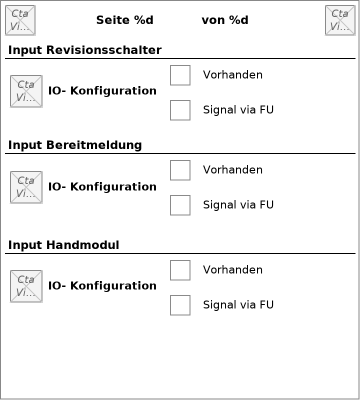
VISUALIZATION VIS_VERDICHTER_PARAMETER_IO  // 360x400
VAR_INPUT
    ITF_VERDICHTERIN : ITF_VERDICHTER;
END_VAR
VAR
    uiPage  :   UINT;
    uiMin   :   UINT    := 0;
    uiMax   :   UINT    := 4
;
END_VAR
    Frame (0,40 360x360), frame switch variable: uiPage
        shows VIS_VERDICHTER_PARAMETER_IO0(ITF_VERDICHTERIN := ITF_VERDICHTERIN, ITF_RevSwitch_IN := ITF_VERDICHTERIN.proRevisionSwitch_ITF, ITF_VerdiReady_IN := ITF_VERDICHTERIN.proReady_ITF, ITF_VerdiHandMod_IN := ITF_VERDICHTERIN.proHandModul_ITF)
        shows VIS_VERDICHTER_PARAMETER_IO1(ITF_VERDICHTERIN := ITF_VERDICHTERIN, ITF_VerdichterOn_IN := ITF_VERDICHTERIN.proIsOn_ITF)
        shows VIS_VERDICHTER_PARAMETER_IO2(ITF_VERDICHTERIN := ITF_VERDICHTERIN, ITF_VerdiNoError_IN := ITF_VERDICHTERIN.proNoError_ITF)
        shows VIS_VERDICHTER_PARAMETER_IO3(ITF_VERDICHTERIN := ITF_VERDICHTERIN, ITF_ActualValue_IN := ITF_VERDICHTERIN.proActualValue_ITF)
        shows VIS_VERDICHTER_PARAMETER_IO4(ITF_VERDICHTERIN := ITF_VERDICHTERIN, ITF_xOn_IN := ITF_VERDICHTERIN.proOn_ITF, ITF_rOnY_IN := ITF_VERDICHTERIN.proOnY_ITF)
    Image (325,5 30x30), invisible if: uiPage = uiMax, image: CtaVisSymbols.ImagePool.arrow-right_square
        OnMouseClick: execute {
            uiPage := uiPage + 1;
            IF uiPage >= uiMax THEN
                uiPage := uiMax;
            END_IF;
        }
    Image (5,5 30x30), invisible if: uiPage = uiMin, image: CtaVisSymbols.ImagePool.arrow-left_square
        OnMouseClick: execute {
            uiPage := uiPage - 1;
            IF uiPage <= uiMin THEN
                uiPage := uiMin;
            END_IF;
        }
    Textfield (175,5 100x30), "von %d", text variable: uiMax
    Textfield (75,5 100x30), "Seite %d", text variable: uiPage
END_VISUALIZATION

// 40 Visualizations/POPUP/PARAMETER/VERDICHTER_IO/VIS_VERDICHTER_PARAMETER_IO2
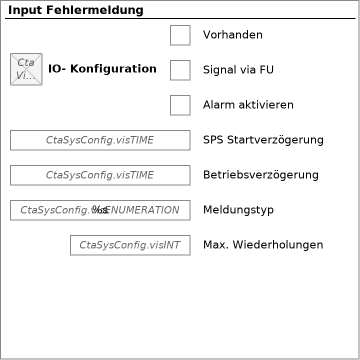
VISUALIZATION VIS_VERDICHTER_PARAMETER_IO2  // 360x360
VAR_INPUT
    ITF_VERDICHTERIN 		:	ITF_VERDICHTER;
	ITF_VerdiNoError_IN		:	CtaSysIO.ITF_IO;
END_VAR
    Label (5,0 350x20), "Input Fehlermeldung"
    Frame (170,25 20x20)
        shows CtaSysConfig.visBOOL(visfbBOOLIn := ITF_VERDICHTERIN.P_scIO_IsNoError_fbxEnable)
    Label (200,25 150x20), "Vorhanden"
    Frame (170,60 20x20)
        shows CtaSysConfig.visBOOL(visfbBOOLIn := ITF_VERDICHTERIN.P_scIO_IsNoError_fbxInputMb)
    Label (200,60 150x20), "Signal via FU"
    Frame (170,95 20x20)
        shows CtaSysConfig.visBOOL(visfbBOOLIn := ITF_VERDICHTERIN.P_scIO_IsNoError_fbxDoesAlarm)
    Label (200,95 150x20), "Alarm aktivieren"
    Frame (10,130 180x20)
        shows CtaSysConfig.visTIME(visfbTIMEIn := ITF_VERDICHTERIN.P_scIO_IsNoError_fbtDelayStartSps)
    Label (200,130 150x20), "SPS Startverzögerung"
    Label (200,165 150x20), "Betriebsverzögerung"
    Frame (10,165 180x20)
        shows CtaSysConfig.visTIME(visfbTIMEIn := ITF_VERDICHTERIN.P_scIO_IsNoError_fbtDelayRun)
    Label (200,200 150x20), "Meldungstyp"
    Label (200,235 150x20), "Max. Wiederholungen"
    Line (5,18) (355,18)
    Frame (70,235 120x20)
        shows CtaSysConfig.visINT(visfbINTIn := ITF_VERDICHTERIN.P_scIO_IsNoError_fbiMaxErrorRetryAllowed)
    Frame (10,200 180x20)
        shows CtaSysConfig.visENUMERATION(visfbENUIn := ITF_VERDICHTERIN.P_scIO_IsNoError_fbiTypeOfAck)
    Image (10,53 32x32), invisible if: ITF_VerdiNoError_IN = 0, image: CtaVisSymbols.ImagePool.build
        OnMouseDown:  Dialog=VIS_ANTRIEB_POPUP_IO_ITF, Parameters={ITF_IO_IN: ITF_VerdiNoError_IN}, OpenModal=True, OpenCentered=True
    Label (45,59 120x20), "IO- Konfiguration", invisible if: ITF_VerdiNoError_IN = 0
    Textfield (30,200 140x20), "%s", text list: 'CtaAppReport.txtLibAp99_2enTypeOfAck', text index: CtaSysConfig.fcGetEnumerationId(ITF_VERDICHTERIN.P_scIO_IsNoError_fbiTypeOfAck)
END_VISUALIZATION

// 40 Visualizations/POPUP/PARAMETER/VERDICHTER_IO/VIS_VERDICHTER_PARAMETER_IO3
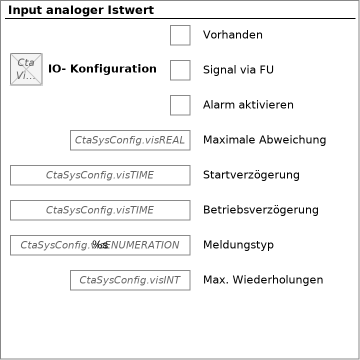
VISUALIZATION VIS_VERDICHTER_PARAMETER_IO3  // 360x360
VAR_INPUT
    ITF_VERDICHTERIN 	:	ITF_VERDICHTER;
	ITF_ActualValue_IN	:	CtaSysIO.ITF_IO;
END_VAR
    Label (5,0 350x20), "Input analoger Istwert"
    Frame (170,25 20x20)
        shows CtaSysConfig.visBOOL(visfbBOOLIn := ITF_VERDICHTERIN.P_scIO_IsValue_fbxEnable)
    Label (200,25 150x20), "Vorhanden"
    Frame (170,60 20x20)
        shows CtaSysConfig.visBOOL(visfbBOOLIn := ITF_VERDICHTERIN.P_scIO_IsValue_fbxInputMb)
    Label (200,60 150x20), "Signal via FU"
    Frame (170,95 20x20)
        shows CtaSysConfig.visBOOL(visfbBOOLIn := ITF_VERDICHTERIN.P_scIO_IsValue_fbxDoesAlarm)
    Label (200,95 150x20), "Alarm aktivieren"
    Frame (10,165 180x20)
        shows CtaSysConfig.visTIME(visfbTIMEIn := ITF_VERDICHTERIN.P_scIO_IsValue_fbtDelayStart)
    Label (200,165 150x20), "Startverzögerung"
    Label (200,200 150x20), "Betriebsverzögerung"
    Frame (10,200 180x20)
        shows CtaSysConfig.visTIME(visfbTIMEIn := ITF_VERDICHTERIN.P_scIO_IsValue_fbtDelayRun)
    Frame (70,130 120x20)
        shows CtaSysConfig.visREAL(visfbREALIn := ITF_VERDICHTERIN.P_scIO_IsValue_fbrMaxDiff)
    Label (200,130 150x20), "Maximale Abweichung"
    Label (200,235 150x20), "Meldungstyp"
    Label (200,270 150x20), "Max. Wiederholungen"
    Line (5,18) (355,18)
    Frame (70,270 120x20)
        shows CtaSysConfig.visINT(visfbINTIn := ITF_VERDICHTERIN.P_scIO_IsValue_fbiMaxErrorRetryAllowed)
    Frame (10,235 180x20)
        shows CtaSysConfig.visENUMERATION(visfbENUIn := ITF_VERDICHTERIN.P_scIO_IsValue_fbiTypeOfAck)
    Image (10,53 32x32), invisible if: ITF_ActualValue_IN = 0, image: CtaVisSymbols.ImagePool.build
        OnMouseDown:  Dialog=VIS_ANTRIEB_POPUP_IO_ITF, Parameters={ITF_IO_IN: ITF_ActualValue_IN}, OpenModal=True, OpenCentered=True
    Label (45,59 120x20), "IO- Konfiguration", invisible if: ITF_ActualValue_IN = 0
    Textfield (30,235 140x20), "%s", text list: 'CtaAppReport.txtLibAp99_2enTypeOfAck', text index: CtaSysConfig.fcGetEnumerationId(ITF_VERDICHTERIN.P_scIO_IsValue_fbiTypeOfAck)
END_VISUALIZATION

// 40 Visualizations/POPUP/PARAMETER/VERDICHTER_InfluxDb/VIS_VERDICHTER_PARAMETER_TRENDLOG
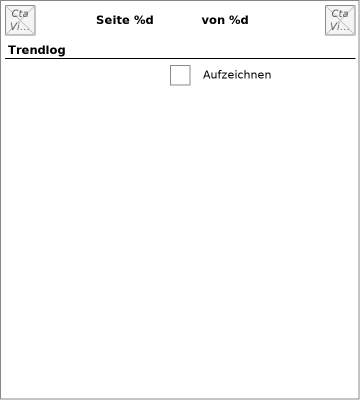
VISUALIZATION VIS_VERDICHTER_PARAMETER_TRENDLOG  // 360x400
VAR_INPUT
    ITF_VERDICHTERIN : ITF_VERDICHTER;
END_VAR
VAR
    uiPage  :   UINT;
    uiMin   :   UINT    := 0;
    uiMax   :   UINT    := 0;
END_VAR
    Image (5,5 30x30), invisible if: uiPage = uiMin, image: CtaVisSymbols.ImagePool.arrow-left_square
        OnMouseClick: execute {
            uiPage := uiPage - 1;
            IF uiPage <= uiMin THEN
                uiPage := uiMin;
            END_IF;
        }
    Image (325,5 30x30), invisible if: uiPage = uiMax, image: CtaVisSymbols.ImagePool.arrow-right_square
        OnMouseClick: execute {
            uiPage := uiPage + 1;
            IF uiPage >= uiMax THEN
                uiPage := uiMax;
            END_IF;
        }
    Frame (0,40 360x360), frame switch variable: uiPage
        shows VIS_VERDICHTER_PARAMETER_TRENDLOG0(ITF_VERDICHTERIN := ITF_VERDICHTERIN)
        shows AT_ParameterIO1(ITF_Parameter := ITF_Parameter)
        pReferences[0]: ITF_Parameter=ITF_Parameter
    Textfield (75,5 100x30), "Seite %d", text variable: uiPage
    Textfield (175,5 100x30), "von %d", text variable: uiMax
END_VISUALIZATION

// 40 Visualizations/POPUP/PARAMETER/VERDICHTER_InfluxDb/VIS_VERDICHTER_PARAMETER_TRENDLOG0
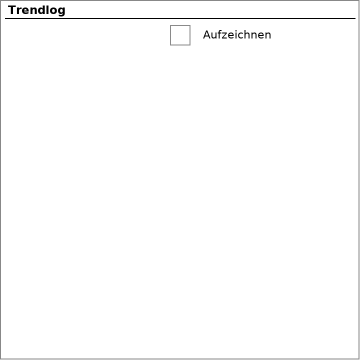
VISUALIZATION VIS_VERDICHTER_PARAMETER_TRENDLOG0  // 360x360
VAR_INPUT
    ITF_VERDICHTERIN : ITF_VERDICHTER;
END_VAR
    Frame (170,25 20x20)
        shows CtaSysConfig.visBOOL(visfbBOOLIn := ITF_VERDICHTERIN.P_scInfluxDb_fbxEnable)
    Label (200,25 150x20), "Aufzeichnen"
    Label (5,0 350x20), "Trendlog"
    Line (5,18) (355,18)
END_VISUALIZATION

// 40 Visualizations/POPUP/IO/VIS_VERDICHTER_IO0
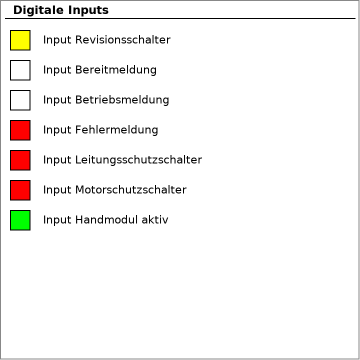
VISUALIZATION VIS_VERDICHTER_IO0  // 360x360
VAR_INPUT
    ITF_VERDICHTERIN    :   ITF_VERDICHTER;	
END_VAR
    Label (40,30 320x20), "Input Revisionsschalter", invisible if: ITF_VERDICHTERIN.proNotShowDI_RevisionSwitchOk
    Label (40,60 320x20), "Input Bereitmeldung", invisible if: ITF_VERDICHTERIN.proNotShowDI_Ready
    Rectangle (10,30 20x20), colour toggle: ITF_VERDICHTERIN.proGetDI_RevisionSwitchOK, invisible if: ITF_VERDICHTERIN.proNotShowDI_RevisionSwitchOk
    Rectangle (10,60 20x20), colour toggle: ITF_VERDICHTERIN.proGetDI_IsReady, invisible if: ITF_VERDICHTERIN.proNotShowDI_Ready
    Label (40,120 320x20), "Input Fehlermeldung", invisible if: ITF_VERDICHTERIN.proNotShowDI_NoError
    Rectangle (10,120 20x20), colour toggle: ITF_VERDICHTERIN.proGetDI_NoError, invisible if: ITF_VERDICHTERIN.proNotShowDI_NoError
    Rectangle (10,150 20x20), colour toggle: ITF_VERDICHTERIN.proGetDI_FuseOK, invisible if: ITF_VERDICHTERIN.proNotShowDI_FuseOk
    Label (40,150 320x20), "Input Leitungsschutzschalter", invisible if: ITF_VERDICHTERIN.proNotShowDI_FuseOk
    Label (40,180 320x20), "Input Motorschutzschalter", invisible if: ITF_VERDICHTERIN.proNotShowDI_VerdichterFuseOk
    Rectangle (10,180 20x20), colour toggle: ITF_VERDICHTERIN.proGetDI_VerdichterFuseOk, invisible if: ITF_VERDICHTERIN.proNotShowDI_VerdichterFuseOk
    Label (40,210 320x20), "Input Handmodul aktiv", invisible if: ITF_VERDICHTERIN.proNotShowDI_VerdichterHand
    Rectangle (10,210 20x20), colour toggle: ITF_VERDICHTERIN.proGetDI_VerdichterHand, invisible if: ITF_VERDICHTERIN.proNotShowDI_VerdichterHand
    Label (40,90 320x20), "Input Betriebsmeldung", invisible if: ITF_VERDICHTERIN.proNotShowDI_IsOn
    Rectangle (10,90 20x20), colour toggle: ITF_VERDICHTERIN.proGetDI_IsOn, invisible if: ITF_VERDICHTERIN.proNotShowDI_IsOn
    Label (10,0 350x20), "Digitale Inputs"
    Line (5,18) (355,18)
END_VISUALIZATION

// 40 Visualizations/POPUP/IO/VIS_VERDICHTER_IO
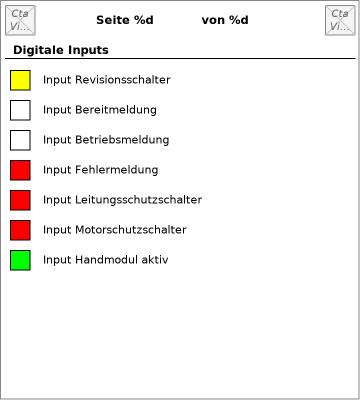
VISUALIZATION VIS_VERDICHTER_IO  // 360x400
VAR_INPUT
    ITF_VERDICHTERIN    :   ITF_VERDICHTER;	
END_VAR
VAR
    uiPage  :   UINT;
    uiMin   :   UINT    := 0;
    uiMax   :   UINT    := 1;
END_VAR
    Frame (0,40 360x360), frame switch variable: uiPage
        shows VIS_VERDICHTER_IO0(ITF_VERDICHTERIN := ITF_VERDICHTERIN)
        shows VIS_VERDICHTER_IO1(ITF_VERDICHTERIN := ITF_VERDICHTERIN)
        shows AT_ParameterIO2(ITF_Parameter := ITF_Parameter)
        shows AT_ParameterIO3(ITF_Parameter := ITF_Parameter)
    Image (325,5 30x30), invisible if: uiPage = uiMax, image: CtaVisSymbols.ImagePool.arrow-right_square
        OnMouseClick: execute {
            uiPage := uiPage + 1;
            IF uiPage >= uiMax THEN
                uiPage := uiMax;
            END_IF;
        }
    Image (5,5 30x30), invisible if: uiPage = uiMin, image: CtaVisSymbols.ImagePool.arrow-left_square
        OnMouseClick: execute {
            uiPage := uiPage - 1;
            IF uiPage <= uiMin THEN
                uiPage := uiMin;
            END_IF;
        }
    Textfield (175,5 100x30), "von %d", text variable: uiMax
    Textfield (75,5 100x30), "Seite %d", text variable: uiPage
END_VISUALIZATION

// 40 Visualizations/POPUP/IO/VIS_VERDICHTER_IO1
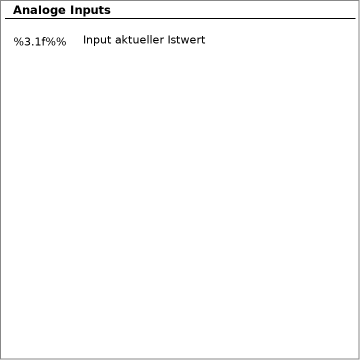
VISUALIZATION VIS_VERDICHTER_IO1  // 360x360
VAR_INPUT
    ITF_VERDICHTERIN    :   ITF_VERDICHTER;	
END_VAR
    Label (80,30 280x20), "Input aktueller Istwert", invisible if: ITF_VERDICHTERIN.proNotShowAI_ActualValue
    Label (10,0 350x20), "Analoge Inputs"
    Textfield (10,32 60x20), "%3.1f%%", text variable: ITF_VERDICHTERIN.proGetAI_ActualValue, invisible if: ITF_VERDICHTERIN.proNotShowAI_ActualValue
    Line (5,18) (355,18)
END_VISUALIZATION

// 40 Visualizations/ICON/VERDICHTER_BASE/VALUE/ValueUpDwn
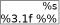
VISUALIZATION ValueUpDwn  // 60x25
VAR_INPUT
    ITF_VERDICHTER_IN   :   ITF_VERDICHTER;	
END_VAR
VAR_INPUT CONSTANT
    uiTextAusrichtung   : UINT := 4;    // 0 = Oben links | 1 = Horizontal zentriert | 2 = Rechts | 4 = Vertikal zentriert | 8 = Unten
END_VAR
    Textfield (0,0 60x12), "%s", text variable: ITF_VERDICHTER_IN.proGetBMK, invisible if: ITF_VERDICHTER_IN.proNoBmkInList
        p3718999670: uiTextAusrichtung
    Textfield (0,13 60x12), "%3.1f %%", text variable: ITF_VERDICHTER_IN.proLeistung, invisible if: NOT ITF_VERDICHTER_IN.proIsRegulatet
        p3718999670: uiTextAusrichtung
END_VISUALIZATION

// 40 Visualizations/ICON/VERDICHTER_LEFT/VERDICHTER_LEFT_ABOVE/VIS_VERDICHTER_LEFT_ABOVE
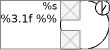
VISUALIZATION VIS_VERDICHTER_LEFT_ABOVE  // 110x50
VAR_INPUT
    ITF_VERDICHTER_IN   :   ITF_VERDICHTER;	
END_VAR
VAR_INPUT CONSTANT
    stExklParameter		:   STRING[40] := '';	
END_VAR
VAR CONSTANT
	uiIconnr		:	UINT := 0;
END_VAR
    Frame (0,0 110x50), invisible if: NOT fcCheckQuerryAndIconReturn(_ITF_IN := ITF_VERDICHTER_IN, _uiIconNr_IN := uiIconNr)
        shows VIS_VERDICHTER_LeftAboveCheckQuerry(ITF_VERDICHTER_IN := ITF_VERDICHTER_IN, stExklParameter := stExklParameter)
END_VISUALIZATION

// 40 Visualizations/ICON/VERDICHTER_LEFT/VERDICHTER_LEFT_ABOVE/VIS_VERDICHTER_LeftAboveCheckIsEnabled
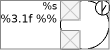
VISUALIZATION VIS_VERDICHTER_LeftAboveCheckIsEnabled  // 110x50
VAR_INPUT
    ITF_VERDICHTER_IN   :   ITF_VERDICHTER;	
    stExklParameter		:   STRING[40];	
END_VAR
    Frame (60,0 50x50), invisible if: NOT ITF_VERDICHTER_IN.proIsEnabled
        shows Icon_Left(ITF_VERDICHTER_IN := ITF_VERDICHTER_IN)
    Frame (0,0 60x25), invisible if: NOT ITF_VERDICHTER_IN.proIsEnabled
        shows ValueUpDwn(ITF_VERDICHTER_IN := ITF_VERDICHTER_IN, uiTextAusrichtung := 6)
    Frame (95,0 15x15), invisible if: NOT ITF_VERDICHTER_IN.proIsEnabled
        shows CommandOn(ITF_VERDICHTER_IN := ITF_VERDICHTER_IN)
    Rectangle (0,0 110x50)
        OnMouseClick:  Dialog=POPUP_VERDICHTER, Parameters={stExklParameter: stExklParameter, ITF_VERDICHTERIN: ITF_VERDICHTER_IN, uiPopUpGruppe: 0}, OpenCentered=True
END_VISUALIZATION

// 40 Visualizations/ICON/VERDICHTER_LEFT/VERDICHTER_LEFT_ABOVE/VIS_VERDICHTER_LeftAboveCheckQuerry
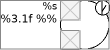
VISUALIZATION VIS_VERDICHTER_LeftAboveCheckQuerry  // 110x50
VAR_INPUT
    ITF_VERDICHTER_IN   :   ITF_VERDICHTER;	
    stExklParameter		:   STRING[40];	
END_VAR
    Frame (0,0 110x50)
        shows VIS_VERDICHTER_LeftAboveCheckIsEnabled(ITF_VERDICHTER_IN := ITF_VERDICHTER_IN, stExklParameter := stExklParameter)
END_VISUALIZATION

// 40 Visualizations/ICON/VERDICHTER_LEFT/VERDICHTER_LEFT_BELOW/VIS_VERDICHTER_LEFT_BELOW
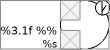
VISUALIZATION VIS_VERDICHTER_LEFT_BELOW  // 110x50
VAR_INPUT
    ITF_VERDICHTER_IN   :   ITF_VERDICHTER;	
END_VAR
VAR_INPUT CONSTANT
    stExklParameter		:   STRING[40] := '';	
END_VAR
VAR CONSTANT
	uiIconNr		:	UINT := 1 ;
END_VAR
    Frame (0,0 110x50), invisible if: NOT fcCheckQuerryAndIconReturn(_ITF_IN := ITF_VERDICHTER_IN, _uiIconNr_IN := uiIconNr)
        shows VIS_VERDICHTER_LeftBelowCheckQuerry(ITF_VERDICHTER_IN := ITF_VERDICHTER_IN, stExklParameter := stExklParameter)
END_VISUALIZATION

// 40 Visualizations/ICON/VERDICHTER_LEFT/VERDICHTER_LEFT_BELOW/VIS_VERDICHTER_LeftBelowCheckIsEnabled
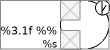
VISUALIZATION VIS_VERDICHTER_LeftBelowCheckIsEnabled  // 110x50
VAR_INPUT
    ITF_VERDICHTER_IN   :   ITF_VERDICHTER;	
    stExklParameter		:   STRING[40];	
END_VAR
    Frame (60,0 50x50), invisible if: NOT ITF_VERDICHTER_IN.proIsEnabled
        shows Icon_Left(ITF_VERDICHTER_IN := ITF_VERDICHTER_IN)
    Frame (0,25 60x27), invisible if: NOT ITF_VERDICHTER_IN.proIsEnabled
        shows ValueDwnUp(ITF_VERDICHTER_IN := ITF_VERDICHTER_IN, uiTextAusrichtung := 6)
    Frame (95,0 15x15), invisible if: NOT ITF_VERDICHTER_IN.proIsEnabled
        shows CommandOn(ITF_VERDICHTER_IN := ITF_VERDICHTER_IN)
    Rectangle (0,0 110x50)
        OnMouseClick:  Dialog=POPUP_VERDICHTER, Parameters={stExklParameter: stExklParameter, ITF_VERDICHTERIN: ITF_VERDICHTER_IN, uiPopUpGruppe: 0}, OpenCentered=True
END_VISUALIZATION

// 40 Visualizations/ICON/VERDICHTER_LEFT/VERDICHTER_LEFT_BELOW/VIS_VERDICHTER_LeftBelowCheckQuerry
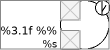
VISUALIZATION VIS_VERDICHTER_LeftBelowCheckQuerry  // 110x50
VAR_INPUT
    ITF_VERDICHTER_IN   :   ITF_VERDICHTER;
    stExklParameter		:   STRING[40];	
END_VAR
    Frame (0,0 110x50)
        shows VIS_VERDICHTER_LeftBelowCheckIsEnabled(ITF_VERDICHTER_IN := ITF_VERDICHTER_IN, stExklParameter := stExklParameter)
END_VISUALIZATION

// 40 Visualizations/ICON/VERDICHTER_RIGHT/VERDICHTER_RIGHT_BELOW/VIS_VERDICHTER_RIGHT_BELOW
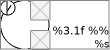
VISUALIZATION VIS_VERDICHTER_RIGHT_BELOW  // 110x50
VAR_INPUT
    ITF_VERDICHTER_IN   :   ITF_VERDICHTER;	
END_VAR
VAR_INPUT CONSTANT
    stExklParameter		:   STRING[40] := '';	
END_VAR
VAR CONSTANT
	uiIconNr		:	UINT := 3;
END_VAR
    Frame (0,0 110x50), invisible if: NOT fcCheckQuerryAndIconReturn(_ITF_IN := ITF_VERDICHTER_IN, _uiIconNr_IN := uiIconNr)
        shows VIS_VERDICHTER_RigthBelowCheckQuerry(ITF_VERDICHTER_IN := ITF_VERDICHTER_IN, stExklParameter := stExklParameter)
END_VISUALIZATION

// 40 Visualizations/ICON/VERDICHTER_RIGHT/VERDICHTER_RIGHT_BELOW/VIS_VERDICHTER_RigthBelowCheckIsEnabled
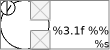
VISUALIZATION VIS_VERDICHTER_RigthBelowCheckIsEnabled  // 110x50
VAR_INPUT
    ITF_VERDICHTER_IN   :   ITF_VERDICHTER;	
    stExklParameter		:   STRING[40];	
END_VAR
    Frame (0,0 50x50), invisible if: NOT ITF_VERDICHTER_IN.proIsEnabled
        shows Icon_Right(ITF_VERDICHTER_IN := ITF_VERDICHTER_IN)
    Frame (52,25 60x27), invisible if: NOT ITF_VERDICHTER_IN.proIsEnabled
        shows ValueDwnUp(ITF_VERDICHTER_IN := ITF_VERDICHTER_IN, uiTextAusrichtung := 4)
    Frame (0,0 15x15), invisible if: NOT ITF_VERDICHTER_IN.proIsEnabled
        shows CommandOn(ITF_VERDICHTER_IN := ITF_VERDICHTER_IN)
    Rectangle (0,0 110x50)
        OnMouseClick:  Dialog=POPUP_VERDICHTER, Parameters={stExklParameter: stExklParameter, ITF_VERDICHTERIN: ITF_VERDICHTER_IN, uiPopUpGruppe: 0}, OpenCentered=True
END_VISUALIZATION

// 40 Visualizations/ICON/VERDICHTER_RIGHT/VERDICHTER_RIGHT_BELOW/VIS_VERDICHTER_RigthBelowCheckQuerry
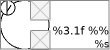
VISUALIZATION VIS_VERDICHTER_RigthBelowCheckQuerry  // 110x50
VAR_INPUT
    ITF_VERDICHTER_IN   :   ITF_VERDICHTER;	
    stExklParameter		:   STRING[40];	
END_VAR
    Frame (0,0 110x50)
        shows VIS_VERDICHTER_RigthBelowCheckIsEnabled(ITF_VERDICHTER_IN := ITF_VERDICHTER_IN, stExklParameter := stExklParameter)
END_VISUALIZATION

// 40 Visualizations/ICON/VERDICHTER_BASE/ICON/Icon_Right
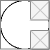
VISUALIZATION Icon_Right  // 50x50
VAR_INPUT
    ITF_VERDICHTER_IN   :   ITF_VERDICHTER;	
END_VAR
    Ellipse (0,0 49x49), colour toggle: ITF_VERDICHTER_IN.proMotorIsOn, invisible if: ITF_VERDICHTER_IN.proIsError
    Ellipse (0,0 49x49), colour toggle: ITF_VERDICHTER_IN.proIsError
    Image (30,0 20x20), invisible if: NOT ITF_VERDICHTER_IN.proIsWarning, image: CtaVisSymbols.ImagePool.CtaWarning
    Image (30,30 20x20), invisible if: NOT ITF_VERDICHTER_IN.proIsHandOnOrOff, image: CtaVisSymbols.ImagePool.front_hand_Yellow
    Image (30,30 20x20), invisible if: NOT ITF_VERDICHTER_IN.proHandOff, image: CtaVisSymbols.ImagePool.front_hand_Yellow_Off
END_VISUALIZATION

// 40 Visualizations/POPUP/PARAMETER/VIS_ANTRIEB_POPUP_IO_ITF
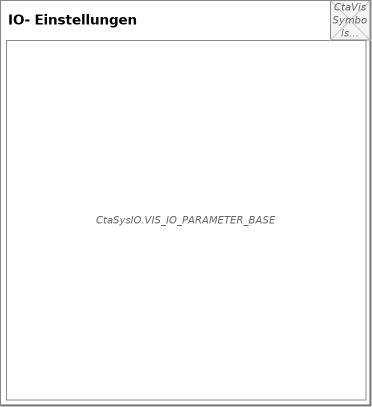
VISUALIZATION VIS_ANTRIEB_POPUP_IO_ITF  // 372x407
VAR_INPUT
    ITF_IO_IN    :   CtaSysIO.ITF_IO;	
END_VAR
    RoundedRectangle (0,0 370x405)
    Frame (6,40 360x360)
        shows CtaSysIO.VIS_IO_PARAMETER_BASE(ITF_IO_IN := ITF_IO_IN)
        shows VIS_ANTRIEB_PARAMETER_IO1(ITF_ANTRIEBIN := ITF_ANTRIEBIN)
        shows VIS_ANTRIEB_PARAMETER_IO2(ITF_ANTRIEBIN := ITF_ANTRIEBIN)
        shows VIS_ANTRIEB_PARAMETER_IO3(ITF_ANTRIEBIN := ITF_ANTRIEBIN)
    Image (330,0 40x40), image: CtaVisSymbols.ImagePool.close_solo_black
        OnMouseClick:  Dialog=VIS_ANTRIEB_POPUP_IO_ITF, Result=None, NumpadKeypadSet=True
    Label (5,0 150x40), "IO- Einstellungen"
END_VISUALIZATION

// 40 Visualizations/POPUP/PARAMETER/VERDICHTER_IO/VIS_VERDICHTER_PARAMETER_IO4
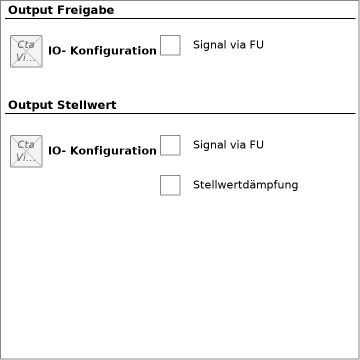
VISUALIZATION VIS_VERDICHTER_PARAMETER_IO4  // 360x360
VAR_INPUT
    ITF_VERDICHTERIN   	:   ITF_VERDICHTER;	
	ITF_xOn_IN			:	CtaSysIO.ITF_IO;
	ITF_rOnY_IN			:	CtaSysIO.ITF_IO;
END_VAR
    Label (5,0 350x20), "Output Freigabe"
    Label (5,95 350x20), "Output Stellwert"
    Line (5,113) (355,113)
    Line (5,18) (355,18)
    Image (10,35 32x32), invisible if: ITF_xOn_IN = 0, image: CtaVisSymbols.ImagePool.build
        OnMouseDown:  Dialog=VIS_ANTRIEB_POPUP_IO_ITF, Parameters={ITF_IO_IN: ITF_xOn_IN}, OpenModal=True, OpenCentered=True
    Image (10,135 32x32), invisible if: ITF_rOnY_IN = 0, image: CtaVisSymbols.ImagePool.build
        OnMouseDown:  Dialog=VIS_ANTRIEB_POPUP_IO_ITF, Parameters={ITF_IO_IN: ITF_rOnY_IN}, OpenModal=True, OpenCentered=True
    Label (45,41 120x20), "IO- Konfiguration", invisible if: ITF_xOn_IN = 0
    Label (45,141 120x20), "IO- Konfiguration", invisible if: ITF_rOnY_IN = 0
    Frame (160,35 20x20)
        shows CtaSysConfig.visBOOL(visfbBOOLIn := ITF_VERDICHTERIN.P_scFU_fbxReleaseMb)
    Label (190,35 150x20), "Signal via FU"
    Frame (160,135 20x20)
        shows CtaSysConfig.visBOOL(visfbBOOLIn := ITF_VERDICHTERIN.P_scFU_fbxSollWertMb)
    Label (190,135 150x20), "Signal via FU"
    Label (190,175 150x20), "Stellwertdämpfung"
    Frame (160,175 20x20)
        shows CtaAppDumper.VisDumperSmall(fbDumper := ITF_VERDICHTERIN.proRefToRonYDumper)
END_VISUALIZATION

// 40 Visualizations/POPUP/OVERVIEW/ResetVerdiTime
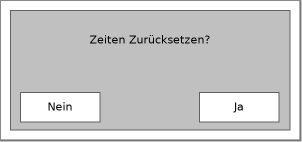
VISUALIZATION ResetVerdiTime  // 302x142
VAR_IN_OUT
	ITF_VERDICHTER_IN		:		ITF_VERDICHTER;
END_VAR
    RoundedRectangle (0,0 300x140)
    RoundedRectangle (10,10 280x120)
    Label (50,10 200x60), "Zeiten Zurücksetzen?"
    RoundedRectangle (20,92 80x30), "Nein"
        OnMouseClick:  Dialog=Current Dialog, Result=None, NumpadKeypadSet=True
    RoundedRectangle (199,92 80x30), "Ja"
        tap ITF_VERDICHTER_IN.proResetVerdiTime
        OnMouseClick:  Dialog=Current Dialog, Result=OK, NumpadKeypadSet=True
END_VISUALIZATION

// 40 Visualizations/POPUP/BUS/VERDICHTER_BUS_SW3_Detail
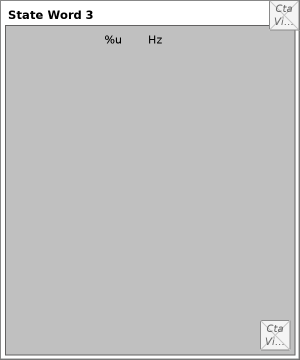
VISUALIZATION VERDICHTER_BUS_SW3_Detail  // 300x360
VAR_IN_OUT
    wDetail             :   WORD;
END_VAR
VAR_INPUT	
    ITF_VERDICHTERIN       :   ITF_VERDICHTER;
END_VAR
VAR_IN_OUT
    xShow               :   BOOL;
END_VAR
    RoundedRectangle (0,0 300x360)
    RoundedRectangle (5,25 290x330)
    Image (269,0 30x30), image: CtaVisSymbols.ImagePool.close_solo_black
        OnMouseClick: execute { xShow := FALSE; ITF_VERDICHTERIN.proModbusTest := FALSE; }
    Label (5,0 150x30), "State Word 3"
    Label (145,30 120x20), "Hz"
    Textfield (15,30 110x20), "%u", text variable: wDetail, input disabled if: NOT ITF_VERDICHTERIn.proModbusTest
        OnMouseClick: write the text variable via InputWithLimits, min 0, max 100
    Textfield (15,30 110x20), "%u", text variable: wDetail, invisible if: ITF_VERDICHTERIN.proModbusTest
    Image (260,320 30x30), invisible if: ITF_VERDICHTERIN.proModbusTest, image: CtaVisSymbols.ImagePool.front_hand_Black
        OnMouseClick: execute { ITF_VERDICHTERIN.proModbusTest := TRUE; }
    Image (260,320 30x30), invisible if: NOT ITF_VERDICHTERIN.proModbusTest, image: CtaVisSymbols.ImagePool.front_hand_Yellow
        OnMouseClick: execute { ITF_VERDICHTERIN.proModbusTest := False; }
END_VISUALIZATION

// 40 Visualizations/ICON/VERDICHTER_BASE/VALUE/ValueDwnUp
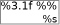
VISUALIZATION ValueDwnUp  // 60x25
VAR_INPUT
    ITF_VERDICHTER_IN   :   ITF_VERDICHTER;	
END_VAR
VAR_INPUT CONSTANT
    uiTextAusrichtung   : UINT := 4;    // 0 = Oben links | 1 = Horizontal zentriert | 2 = Rechts | 4 = Vertikal zentriert | 8 = Unten
END_VAR
    Textfield (0,13 60x12), "%s", text variable: ITF_VERDICHTER_IN.proGetBMK, invisible if: ITF_VERDICHTER_IN.proNoBmkInList
        p3718999670: uiTextAusrichtung
    Textfield (0,0 60x12), "%3.1f %%", text variable: ITF_VERDICHTER_IN.proLeistung, invisible if: NOT ITF_VERDICHTER_IN.proIsRegulatet
        p3718999670: uiTextAusrichtung
END_VISUALIZATION

(* text list Error (id | default | de | en | fr | it)
  0 | keine Meldung Anstehend | Keine Meldung Anstehend | No message pending | Aucun message en attente | Nessun messaggio in sospeso
  1 | keine Betriebsrückmeldung | Keine Betriebsrückmeldung | No operational feedback | Aucune rétroaction opérationnelle | Nessun feedback operativo
  2 | Alarmkontakt Anstehend | Alarmkontakt Anstehend | Error contact pending | Contact d'alarme en attente | Contatto di allarme in sospeso
  3 | Leitungsschutzschalter ausfall | Leitungsschutzschalter ausfall | Circuit breaker failure | Défaillance du disjoncteur | Guasto dell'interruttore
  4 | Motorschutzschalter ausfall | Motorschutzschalter ausfall | Motor protection switch failure | Défaillance de l'interrupteur de protection du moteur | Guasto al salvamotore
  5 | Konfigurationsfehler speichern fehlgeschlagen reboot | Konfigurationsfehler speichern fehlgeschlagen reboot | Failed to save configuration error reboot | Impossible d'enregistrer l'erreur de configuration reboot | Impossibile salvare l'errore di configurazione reboot
   |  |  |  |  |  *)

(* text list Info (id | default | de | en | fr | it)
  0 | keine Meldung Anstehend | keine Meldung Anstehend | no message pending | aucun message en attente | nessun messaggio in sospeso
   |  |  |  |  |  *)

(* text list Warnung (id | default | de | en | fr | it)
  0 | Keine Meldung Anstehend | Keine Meldung Anstehend | No message pending | Aucun message en attente | Nessun messaggio in sospeso
  4 | Wahlschalter Hand, Ein | Wahlschalter Hand, Ein | Selector switch hand on | Commutateur de sélection a main, Allumé | Selettore a mano, acceso
  3 | Wahlschalter Hand, Aus | Wahlschalter Hand, Aus | Selector switch hand off | Commutateur de sélection a main, Éteint | Selettore a mano, spento
  2 | Revisionsschalter Ausgeschalten | Revisionsschalter Ausgeschalten | Revision switch off | Commutateur révision Désactiver | Interruttore di revisione disattivato
  1 | Sicherheits Stopp | Sicherheits Stopp | Safety stop | Arrêt de sécurité | Sosta di sicurezza
  5 | Handmodul aktiv | Handmodul aktiv | Hand module active | Module manuel actif | Modulo manuale attivo
   |  |  |  |  |  *)
